// TIA Portal V20 export
TYPE "LER_typeWeightCheckTrackingData"
// stored: Access Published
   STRUCT
      resultData { ExternalWritable := 'False'} : Real;
      resultOK { ExternalWritable := 'False'} : Bool;
      resultNG { ExternalWritable := 'False'} : Bool;
      complete { ExternalWritable := 'False'} : Bool;
   END_STRUCT;
END_TYPE
